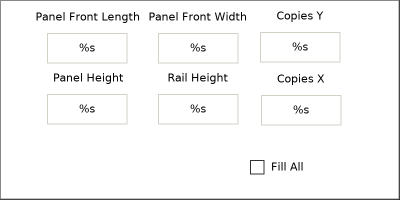
VISUALIZATION V_ProductionBorgoWings  // 400x200
VAR_IN_OUT
	HMI : ST_PackMLBaseModule_HMI;
	HMI_GantryXYZ : ST_GantryXYZ_HMI;
	HMI_Recipe : ST_RecipeBuilder_HMI;
END_VAR
    RoundedRectangle (0,0 400x200)
    Textfield (47,33 80x30), "%s", text variable: HMI_Recipe.Config.PanelFrontLength
        OnMouseClick: write the text variable via VisuDialogs.Numpad, min HMI_Recipe.Limits.PanelFrontLength.MinVal, max HMI_Recipe.Limits.PanelFrontLength.MaxVal
    Label (30,7 116x20), "Panel Front Length"
    Textfield (158,33 80x30), "%s", text variable: HMI_Recipe.Config.PanelFrontWidth
        OnMouseClick: write the text variable via VisuDialogs.Numpad, min HMI_Recipe.Limits.PanelFrontWidth.MinVal, max HMI_Recipe.Limits.PanelFrontWidth.MaxVal
    Label (109,7 178x20), "Panel Front Width"
    Textfield (47,94 80x30), "%s", text variable: HMI_Recipe.Config.PanelHeight
        OnMouseClick: write the text variable via VisuDialogs.Numpad, min HMI_Recipe.Limits.PanelHeight.MinVal, max HMI_Recipe.Limits.PanelHeight.MaxVal
    Label (31,68 115x20), "Panel Height"
    Textfield (158,94 80x30), "%s", text variable: HMI_Recipe.Config.RailHeightCorrection
        OnMouseClick: write the text variable via VisuDialogs.Numpad, min HMI_Recipe.Limits.RailHeightCorrection.MinVal, max HMI_Recipe.Limits.RailHeightCorrection.MaxVal
    Label (147,68 102x20), "Rail Height"
    Checkbox (248,152 72x30), "Fill All", variable: HMI_Recipe.Config.FillAll
    Textfield (261,95 80x30), "%s", text variable: HMI_Recipe.Config.RequestedCopiesX, input disabled if: MAIN.Seedra.RecipeConfig_HMI.Config.FillAll
        OnMouseClick: write the text variable via VisuDialogs.Numpad, min 1, max MAIN.Seedra.RecipeConfig_HMI.Limits.RequestedCopiesX.MaxVal
    Label (250,69 102x20), "Copies X"
    Textfield (260,32 80x30), "%s", text variable: HMI_Recipe.Config.RequestedCopiesY, input disabled if: MAIN.Seedra.RecipeConfig_HMI.Config.FillAll
        OnMouseClick: write the text variable via VisuDialogs.Numpad, min 1, max MAIN.Seedra.RecipeConfig_HMI.Limits.RequestedCopiesY.MaxVal
    Label (249,6 102x20), "Copies Y"
END_VISUALIZATION

(* stored: Version 1.1.0.1, ProductVersion 3.1.4024.15
   Visu V_ProductionBorgoWings: Id {efad271e-12d1-4fb0-b506-e59d88a07246} *)
